# EPICS autosave request: mw100App/Db/MW100_relay_slot3_settings.req
$(P)$(DAU):021:Label
$(P)$(DAU):022:Label
$(P)$(DAU):023:Label
$(P)$(DAU):024:Label
$(P)$(DAU):025:Label
$(P)$(DAU):026:Label
$(P)$(DAU):027:Label
$(P)$(DAU):028:Label
$(P)$(DAU):029:Label
$(P)$(DAU):030:Label
